FUNCTION_BLOCK FB_CalcXRayAbsorptionConstantMock EXTENDS FB_FalliblePublicMock IMPLEMENTS I_CalcXRayAbsorptionConstant
VAR
    fbResult : FB_QuantityLREALPublic(Units := '1');
END_VAR


METHOD Calculate
VAR_INPUT
    MaterialFormula	: T_MaxString;
    AbsorptionConstant	: I_QuantityLREALPublic;
END_VAR

AbsorptionConstant.Copy(fbResult);
END_METHOD


METHOD SetResult
VAR_INPUT
    Result : I_QuantityLREAL;
END_VAR

fbResult.Copy(QuantityToCopy := Result);
END_METHOD


METHOD SetValid

fbResult.Val := 1.0;
fbResult.Units := '1/m';
fbResult.ClearError();
ClearError();
END_METHOD

END_FUNCTION_BLOCK

(* stored: Version 1.1.0.1
   POU FB_CalcXRayAbsorptionConstantMock: Id {b5e25519-ff34-4705-a41c-07a33cb4f6f6}, SpecialFunc None
   Method Calculate: Id {94aba10b-275d-4077-b728-766a54da529d}
   Method SetResult: Id {94d86c85-0b5e-4065-b511-44934c8eb565}
   Method SetValid: Id {afb99497-16bd-4be9-baa6-a37f9f34dc80} *)
